// TwinCAT 3 PLC project MachineA
// ProgramVersion: 3.1.4023.0
// libraries:
//   Tc2_Standard, * (Beckhoff Automation GmbH)
//   Tc2_System, * (Beckhoff Automation GmbH)
//   Tc3_Module, * (Beckhoff Automation GmbH)
// project tree:
//   02_Machine/ FB_Machine.TcPOU
//   03_Module/Arm/ E_ArmState.TcDUT, FB_Arm.TcPOU
//   04_Component/Inverter/ FB_Inverter.TcPOU
//   04_Component/Sensor/ FB_Sensor.TcPOU
//   / PlcTask.TcTTO
//   01_Application/ MAIN.TcPOU
// real-time tasks:
//   TASK PlcTask: cycle T#10ms, priority 20, ADS port 350
//   TASK PlcTask1: cycle T#10ms, priority 21, ADS port 351

CONFIGURATION MachineA
    RESOURCE PLC ON TwinCAT3
        TASK PlcTask(INTERVAL := T#10ms, PRIORITY := 20);
        PROGRAM MAIN WITH PlcTask : MAIN;
    END_RESOURCE
END_CONFIGURATION

// ---- 03_Module/Arm/E_ArmState.TcDUT
{attribute 'qualified_only'}
{attribute 'strict'}
TYPE E_ArmState :
(
	Idle			:= 0,
	FirstState		:= 1,
	Redo			:= 2,
	SecondState		:= 3,
	Done			:= 4,
	
	Reverse			:= 5,
	Inverse			:= 6
) := Idle;
END_TYPE

// ---- 01_Application/MAIN.TcPOU
PROGRAM MAIN
VAR
	fbMachine				: FB_Machine;
END_VAR

fbMachine();

END_PROGRAM

// ---- 02_Machine/FB_Machine.TcPOU
FUNCTION_BLOCK FB_Machine
VAR
	(*
	fbArm				: FB_Arm;
	
	(*Arm*)
		(*Button*)
	btStartHoming		: BOOL;
	btStartPositioning	: BOOL;
	
		(*Set*)
	rHighSpeedHzValue	: REAL;
	rLowSpeedHzValue	: REAL;
	rHzToRawRatioValue	: REAL;
	tDelayTimeValue		: TIME;
	
	rTargetAxis			: REAL;
		(*Get*)
	rCurAxis			: REAL;
	*)
END_VAR

(*
fbArm.HighSpeedHz := rHighSpeedHzValue;
fbArm.LowSpeedHz := rLowSpeedHzValue;
fbArm.HzToRawRatio := rHzToRawRatioValue;
fbArm.DelayTime := tDelayTimeValue;

IF fbArm.Homing(btStartHoming) THEN
	btStartHoming := FALSE;
END_IF

IF fbArm.Positioning(btStartPositioning, rTargetAxis) THEN
	btStartPositioning := FALSE;
END_IF
*)

Arm();

METHOD Arm : PVOID
VAR
	fbArm				: FB_Arm;
	
	(*Arm*)
		(*Button*)
	btStartHoming		: BOOL;
	btStartPositioning	: BOOL;
	
		(*Set*)
	rHighSpeedHzValue	: REAL;
	rLowSpeedHzValue	: REAL;
	rHzToRawRatioValue	: REAL;
	tDelayTimeValue		: TIME;
	
	rTargetAxis			: REAL;
		(*Get*)
	rCurAxis			: REAL;
END_VAR
fbArm.HighSpeedHz := rHighSpeedHzValue;
fbArm.LowSpeedHz := rLowSpeedHzValue;
fbArm.HzToRawRatio := rHzToRawRatioValue;
fbArm.DelayTime := tDelayTimeValue;

IF fbArm.Homing(btStartHoming) THEN
	btStartHoming := FALSE;
END_IF

IF fbArm.Positioning(btStartPositioning, rTargetAxis) THEN
	btStartPositioning := FALSE;
END_IF
END_METHOD

END_FUNCTION_BLOCK

// ---- 03_Module/Arm/FB_Arm.TcPOU
FUNCTION_BLOCK FB_Arm
VAR
	fbInverter				: FB_Inverter;
	fbFrontSensor			: FB_Sensor;
	fbHomeSensor			: FB_Sensor;
	fbRearSensor			: FB_Sensor;
	
	(*Arm State*)
	bBusy					: BOOL;
	bHoming					: BOOL;
		iHomingState		: INT;
	bJogging				: BOOL;
	bPositioning			: BOOL;
		iPositioningState	: INT;
	bInverseDirection		: BOOL;
	
	(*Parameter*)
	rHighSpeedHz			: REAL;
	rLowSpeedHz				: REAL;
	rHzToRawRatio			: REAL;
	rAnalog					: REAL;
	tDelayTime				: TIME;
	
	rAxisSV					: REAL;
	rAxisPV					: REAL	:= fbInverter.Axis;
	(*Others*)
	fbTon					: TON;
END_VAR

PROPERTY Axis : REAL
GET
Axis := rAxisPV;
END_GET
END_PROPERTY

PROPERTY DelayTime : TIME
SET
tDelayTime := DelayTime;
END_SET
END_PROPERTY

PROPERTY HighSpeedHz : REAL
SET
rHighSpeedHz := HighSpeedHz;
END_SET
END_PROPERTY

METHOD Homing : BOOL
VAR_INPUT
	StartButton				: BOOL;
END_VAR
CASE iHomingState OF
	E_ArmState.Idle:
		IF StartButton AND NOT bHoming AND NOT bBusy AND NOT fbHomeSensor.Detect THEN
			bBusy := TRUE;
			bHoming := TRUE;
			
			iHomingState := E_ArmState.FirstState;
			
		ELSIF StartButton AND fbHomeSensor.Detect THEN
			iHomingState := E_ArmState.Done;
		END_IF
	
	E_ArmState.FirstState:
			fbInverter.Analog := (rHzToRawRatio*rHighSpeedHz);
		MoveLeft();
		
		IF fbHomeSensor.Detect THEN
			MoveStop();
			
			fbTon(IN:= TRUE, PT:= tDelayTime);
			IF fbTon.Q THEN
				fbTon(IN:= FALSE);
				iHomingState := E_ArmState.Redo;
			END_IF
			
		ELSIF fbFrontSensor.Detect THEN
			MoveStop();
			
			fbTon(IN:= TRUE, PT:= tDelayTime);
			IF fbTon.Q THEN
				fbTon(IN:= FALSE);
				iHomingState := E_ArmState.Reverse;
			END_IF
			
		ELSIF fbRearSensor.Detect THEN
			MoveStop();
			
			fbTon(IN:= TRUE, PT:= tDelayTime);
			IF fbTon.Q THEN
				fbTon(IN:= FALSE);
				bInverseDirection := NOT bInverseDirection;
				iHomingState := E_ArmState.Inverse;
			END_IF
		END_IF
	
	E_ArmState.Reverse:
		MoveRight();
		
		IF fbHomeSensor.Detect THEN
			MoveStop();
			fbTon(IN:= TRUE, PT:= tDelayTime);
			IF fbTon.Q THEN
				fbTon(IN:= FALSE);
				iHomingState := E_ArmState.Redo;
			END_IF
		END_IF
	
	E_ArmState.Inverse:
		MoveLeft();
		
		IF fbHomeSensor.Detect THEN
			MoveStop();
			fbTon(IN:= TRUE, PT:= tDelayTime);
			IF fbTon.Q THEN
				fbTon(IN:= FALSE);
				iHomingState := E_ArmState.Redo;
			END_IF
		END_IF
	
	E_ArmState.Redo:
		fbInverter.Analog := (rHzToRawRatio*rLowSpeedHz);
		MoveLeft();
		
		IF NOT fbHomeSensor.Detect THEN
			MoveStop();
			fbTon(IN:= TRUE, PT:= tDelayTime);
			IF fbTon.Q THEN
				fbTon(IN:= FALSE);
				iHomingState := E_ArmState.SecondState;
			END_IF
		END_IF
	
	E_ArmState.SecondState:
		fbInverter.Analog := (rHzToRawRatio*rLowSpeedHz);
		MoveRight();
		IF fbHomeSensor.Detect THEN
			MoveStop();
			
			fbTon(IN:= TRUE, PT:= tDelayTime);
			IF fbTon.Q THEN
				fbTon(IN:= FALSE);
				iHomingState := E_ArmState.Done;
			END_IF
		END_IF
	
	E_ArmState.Done:
		bBusy := FALSE;
		bHoming := FALSE;
		iHomingState := E_ArmState.Idle;
		Homing := True;
END_CASE
END_METHOD

PROPERTY HzToRawRatio : REAL
SET
rHzToRawRatio := HzToRawRatio;
END_SET
END_PROPERTY

METHOD Jogging : BOOL
VAR_INPUT
	StartButton				: BOOL;
	MoveLeftButton			: BOOL;
	MoveRightButton			: BOOL;
END_VAR
END_METHOD

PROPERTY LowSpeedHz : REAL
SET
rLowSpeedHz := LowSpeedHz;
END_SET
END_PROPERTY

METHOD PRIVATE MoveLeft : PVOID
VAR_INPUT
END_VAR
IF NOT bInverseDirection THEN
	fbInverter.Clockwise := TRUE;
	fbInverter.CounterClockwise := FALSE;
ELSE
	fbInverter.Clockwise := FALSE;
	fbInverter.CounterClockwise := TRUE;
END_IF
END_METHOD

METHOD PRIVATE MoveRight : PVOID
VAR_INPUT
END_VAR
IF NOT bInverseDirection THEN
	fbInverter.Clockwise := FALSE;
	fbInverter.CounterClockwise := TRUE;
ELSE
	fbInverter.Clockwise := TRUE;
	fbInverter.CounterClockwise := FALSE;
END_IF
END_METHOD

METHOD PRIVATE MoveStop : PVOID
VAR_INPUT
END_VAR
fbInverter.Clockwise := FALSE;
fbInverter.CounterClockwise := FALSE;
END_METHOD

METHOD Positioning : BOOL
VAR_INPUT
	StartButton				: BOOL;
	TargetAxis				: REAL;
END_VAR
CASE iPositioningState OF
	E_ArmState.Idle:
		IF StartButton AND NOT bPositioning AND NOT bBusy THEN
			bBusy := TRUE;
			bHoming := TRUE;
			
			iPositioningState := E_ArmState.FirstState;
		END_IF
	
	E_ArmState.FirstState:
		IF fbFrontSensor.Detect OR fbFrontSensor.Detect THEN
			MoveStop();
			
			fbTon(IN:= TRUE, PT:= tDelayTime);
			IF fbTon.Q THEN
				fbTon(IN:= FALSE);
				iPositioningState := E_ArmState.Inverse;
			END_IF
		ELSE
			IF REAL_TO_INT(fbInverter.Axis) < REAL_TO_INT(TargetAxis) THEN
				IF (TargetAxis - fbInverter.Axis) > 10 THEN
					fbInverter.Analog := (rHzToRawRatio*rHighSpeedHz);
				ELSE
					fbInverter.Analog := (rHzToRawRatio*rHighSpeedHz);
				END_IF
				MoveLeft();
				
			ELSIF REAL_TO_INT(fbInverter.Axis) > REAL_TO_INT(TargetAxis) THEN
				IF (fbInverter.Axis - TargetAxis) > 10 THEN
					fbInverter.Analog := (rHzToRawRatio*rHighSpeedHz);
				ELSE
					fbInverter.Analog := (rHzToRawRatio*rHighSpeedHz);
				END_IF
				MoveRight();
			
			ELSE
				MoveStop();
				
				fbTon(IN:= TRUE, PT:= tDelayTime);
				IF fbTon.Q THEN
					fbTon(IN:= FALSE);
					iPositioningState := E_ArmState.Done;
				END_IF
			END_IF
		END_IF
		
	E_ArmState.Inverse:
		MoveLeft();
		
		IF fbHomeSensor.Detect THEN
			MoveStop();
			fbTon(IN:= TRUE, PT:= tDelayTime);
			IF fbTon.Q THEN
				fbTon(IN:= FALSE);
				iPositioningState := E_ArmState.FirstState;
			END_IF
		END_IF
	
	E_ArmState.Done:
		bBusy := FALSE;
		bPositioning := FALSE;
		iPositioningState := E_ArmState.Idle;
		Positioning := TRUE;
END_CASE
END_METHOD

END_FUNCTION_BLOCK

// ---- 04_Component/Inverter/FB_Inverter.TcPOU
FUNCTION_BLOCK FB_Inverter
VAR
	rAnalogSV				AT %Q* : REAL;
	
	rAxisPV					AT %I* : REAL;
	
	bClockwise				AT %Q* : BOOL;
	bCounterClockwise		AT %Q* : BOOL;
	
END_VAR

PROPERTY Analog : REAL
SET
rAnalogSV := Analog;
END_SET
END_PROPERTY

PROPERTY Axis : REAL
GET
Axis := rAxisPV;
END_GET
END_PROPERTY

PROPERTY Clockwise : BOOL
SET
bClockwise := Clockwise;
END_SET
END_PROPERTY

PROPERTY CounterClockwise : BOOL
SET
bCounterClockwise := CounterClockwise;
END_SET
END_PROPERTY

END_FUNCTION_BLOCK

// ---- 04_Component/Sensor/FB_Sensor.TcPOU
FUNCTION_BLOCK FB_Sensor
VAR
	bDetect					AT %I* : BOOL;
END_VAR

PROPERTY Detect : BOOL
GET
Detect := bDetect;
END_GET
END_PROPERTY

END_FUNCTION_BLOCK
